PROGRAM EncoderMeas
VAR
	
encoder1:ENCODERPULSEtoANGLE;
encoder2:ENCODERPULSEtoANGLE;

END_VAR

//Dónde estoy?

//ALFA
///Realidad
IF NOT(GVL.Scarafitti.simulacion_alfa) THEN
////Calibración
encoder1.angulo_calibrado:=GVL.Pi;
encoder1.b_calibrado:=IO.tope_alfa;
////Medir ángulos
encoder1.A:=IO.encoder1_A;
encoder1.B:=IO.encoder1_B;
encoder1();
GVL.alfa:=encoder1.angle;
ELSE
///Simulación
GVL.alfa:=IO.alfa_sim;
END_IF

//BETA
///Realidad
IF NOT(GVL.Scarafitti.simulacion_beta) THEN
////Calibración
encoder2.angulo_calibrado:=0;
encoder2.b_calibrado:=IO.tope_beta;
////Medir ángulos
encoder2.A:=IO.encoder2_A;
encoder2.B:=IO.encoder2_B;
encoder2();
GVL.beta:=encoder2.angle;
ELSE
///Simulación
GVL.beta:=IO.beta_sim;
END_IF

END_PROGRAM

(* stored: Version 1.1.0.1, ProductVersion 3.1.4024.4
   POU EncoderMeas: Id {0d96bc1c-ffb1-440d-b63c-eed900a16197}, SpecialFunc None *)
